INTERFACE I_RoomTemp

PROPERTY nRoomTemp : REAL
GET
END_GET
END_PROPERTY

END_INTERFACE

(* stored: Version 1.1.0.1
   Itf I_RoomTemp: Id {7f258d7a-27bc-4e5b-bac9-670543498c63}
   Property nRoomTemp: Id {e1b4056e-a903-4bcb-85d8-1d188783f658}
   Get Get: Id {c67c22e4-25fc-4bcb-b688-d90eb51c9d53} *)
